// TIA Portal project "MIxProject" (V21)

(* hardware
DEVICE "S7-1500/ET200MP station_1"  S7-1500 station
   slot 0: "Rail_0"  Rack  6ES7 590-1***0-0AA0
   slot 1: "PLC_1"  CPU 1511-1 PN  6ES7 511-1AK02-0AB0  V2.9
      slot 3: "CPU display_1"  6ES7591-1AA00-0AA0
      slot 32768: "PROFINET interface_1"  X1
         slot 32769: "Port_1"  X1 P1
         slot 32770: "Port_2"  X1 P2
      slot 34817: "Virtual CP interface port_1"  Virtual CP interface port  Virtual CP interface port
DEVICE "HMI_1"  KTP700 Basic PN
   slot 0: "HMI_1"  KTP700 Basic PN  6AV2 123-2GB03-0AX0  17.0.0.0
   slot 1: "HMI_RT_1"  KTP700 Basic PN  6AV2 123-2GB03-0AX0  17.0.0.0
   slot 5: "HMI_1.IE_CP_1"  PROFINET Interface  17.0.0.0
      slot 1: "PROFINET Interface_1"  PROFINET Interface
         slot 1: "Port_1"  Port
*)

// ===== PLC "PLC_1"  CPU 1511-1 PN =====

VAR_GLOBAL   // PLC tag table "Default tag table"
   "valveA" AT %Q0.0 : Bool;
   "valveB" AT %Q0.1 : Bool;
   "valveC" AT %Q0.2 : Bool;
   "MIX" AT %Q0.3 : Bool;
   "TempSensor" AT %MD100 : Real;
   "LevelSensor" AT %MD200 : Real;
   "Start" AT %I0.4 : Bool;
   "Stop" AT %I0.5 : Bool;
   "Emergency" AT %I0.6 : Bool;
   "HeaterON/OFF" AT %M0.0 : Bool;
   "HeaterOutput" AT %MD300 : Real;
   "Setpoint" AT %MD4 : Real;
   "CurrentStep" AT %MW400 : Int;
END_VAR

DATA_BLOCK "FB_MixingSequence_DB"   // DB1
{ S7_Optimized_Access := 'TRUE' }
VERSION : 0.1
// stored: InstanceOfName FB_MixingSequence
"FB_MixingSequence"
BEGIN
END_DATA_BLOCK

DATA_BLOCK "sim_DB"   // DB3
{ S7_Optimized_Access := 'TRUE' }
VERSION : 0.1
// stored: InstanceOfName sim
"sim"
BEGIN
END_DATA_BLOCK

FUNCTION_BLOCK "FB_MixingSequence"   // FB1, GRAPH_PLUS
{ S7_Optimized_Access := 'TRUE' }
VERSION : 0.1
   VAR_INPUT
      OFF_SQ : Bool := false;   // Turn sequence off
      INIT_SQ : Bool := false;   // Set sequence to initial state
      ACK_EF : Bool := false;   // Acknowledge all errors and faults
      S_PREV : Bool := false;   // Output previous step in parameter S_NO
      S_NEXT : Bool := false;   // Indicate next step in parameter S_NO
      SW_AUTO : Bool := false;   // Automatic mode
      SW_TAP : Bool := false;   // Semiautomatic/switch with transition
      SW_TOP : Bool := false;   // Semiautomatic/ignore transition
      SW_MAN : Bool := false;   // Manual mode
      S_SEL : Int := 0;   // Select step to be output to S_NO
      S_ON : Bool := false;   // Activate step indicated in S_NO
      S_OFF : Bool := false;   // Disable step indicated in S_NO
      T_PUSH : Bool := false;   // Enable transition to switch in semi automatic mode
   END_VAR
   VAR_OUTPUT
      S_NO : Int := 0;   // Step number
      S_MORE : Bool := false;   // More steps are available and can be shown in S_NO
      S_ACTIVE : Bool := false;   // Step indicated in S_NO is active
      ERR_FLT : Bool := false;   // Interlock or supervision group error
      AUTO_ON : Bool := false;   // Automatic mode is active
      TAP_ON : Bool := false;   // Semiautomatic mode/step with transition enabled
      TOP_ON : Bool := false;   // Semiautomatic mode/ignore transition enabled
      MAN_ON : Bool := false;   // Manual mode is active
   END_VAR
   VAR
      HMI_INFO : Array[0..8] of UInt;
      IF_PAR : G7_IfParPlus_V6;
      RT_DATA : G7_RTDataPlus_V6;   // Internal data area
      Trans1 : G7_TransitionPlus_V6;   // Transition structure
      Trans2 : G7_TransitionPlus_V6;   // Transition structure
      Trans3 : G7_TransitionPlus_V6;   // Transition structure
      Trans4 : G7_TransitionPlus_V6;   // Transition structure
      Trans5 : G7_TransitionPlus_V6;   // Transition structure
      Step1 : G7_StepPlus_V6;   // Step structure
      Step2 : G7_StepPlus_V6;   // Step structure
      Step3 : G7_StepPlus_V6;   // Step structure
      Step4 : G7_StepPlus_V6;   // Step structure
      Step5 : G7_StepPlus_V6;   // Step structure
      SINI : Array[0..1] of USInt;
      LSTT : Array[0..4] of USInt;
      ATAJ : Array[0..4] of USInt;
      ATAB : Array[0..4] of USInt;
      PSTT : Array[0..4] of USInt;
      NSTT : Array[0..4] of USInt;
      ASSJ : Array[0..4] of USInt;
      ASSB : Array[0..4] of USInt;
      PTTS : Array[0..4] of USInt;
      NTTS : Array[0..4] of USInt;
      SW_SQTS : Array[0..4] of USInt;
      SWITCH : Array[0..0] of USInt;
      TVX : Array[0..1] of USInt;
      TTX : Array[0..1] of USInt;
      TSX : Array[0..1] of USInt;
      S00X : Array[0..1] of USInt;
      SOFFX : Array[0..1] of USInt;
      SONX : Array[0..1] of USInt;
      SAX : Array[0..1] of USInt;
      SERRX : Array[0..5] of USInt;
      SMX : Array[0..5] of USInt;
      S0X : Array[0..5] of USInt;
      S1X : Array[0..5] of USInt;
      IL_ALARM_INST : Diag_Alarm;
      SUP_ALARM_INST : Diag_Alarm;
      STEP_TIME_ALARM_INST : Diag_Alarm;
      IEC_TIMER_INST : IEC_TIMER;
      TRANSACTION_FLAG : Bool := false;
   END_VAR
   // SINI[0] := 2;
   // LSTT[0] := 255;
   // LSTT[1] := 255;
   // LSTT[2] := 255;
   // LSTT[3] := 255;
   // ATAJ[1] := 1;
   // ATAJ[2] := 2;
   // ATAJ[3] := 3;
   // ATAJ[4] := 4;
   // ATAB[1] := 1;
   // ATAB[2] := 2;
   // ATAB[3] := 3;
   // ATAB[4] := 4;
   // PSTT[1] := 1;
   // PSTT[2] := 2;
   // PSTT[3] := 3;
   // PSTT[4] := 4;
   // NSTT[0] := 1;
   // NSTT[1] := 2;
   // NSTT[2] := 3;
   // NSTT[3] := 4;
   // ASSJ[1] := 1;
   // ASSJ[2] := 2;
   // ASSJ[3] := 3;
   // ASSJ[4] := 4;
   // ASSB[1] := 1;
   // ASSB[2] := 2;
   // ASSB[3] := 3;
   // ASSB[4] := 4;
   // PTTS[0] := 255;
   // PTTS[2] := 1;
   // PTTS[3] := 2;
   // PTTS[4] := 3;
   // NTTS[1] := 1;
   // NTTS[2] := 2;
   // NTTS[3] := 3;
   // NTTS[4] := 4;
   // TVX[0] := 16#1;
   // TTX[0] := 16#1;
   // TSX[0] := 16#1;
   // S00X[0] := 16#1;
   // SOFFX[0] := 16#1;
   // SONX[0] := 16#1;
   // SAX[0] := 16#1;
   // SERRX[0] := 16#1;
   // SMX[0] := 16#1;
   // S0X[0] := 16#1;
   // S1X[0] := 16#1;
BEGIN
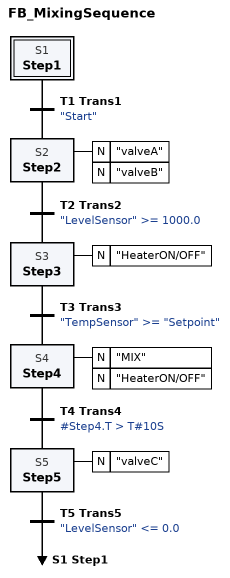
   // sequencer 1
   INITIAL_STEP Step1:   // S1, max time T#10S, warning time T#7S
   END_STEP
   TRANSITION Trans1 FROM Step1 TO Step2   // T1
      := "Start";
   END_TRANSITION
   STEP Step2:   // S2, max time T#10S, warning time T#7S
              N    "valveA"
              N    "valveB"
   END_STEP
   TRANSITION Trans2 FROM Step2 TO Step3   // T2
      := "LevelSensor" >= 1000.0;
   END_TRANSITION
   STEP Step3:   // S3, max time T#10S, warning time T#7S
              N    "HeaterON/OFF"
   END_STEP
   TRANSITION Trans3 FROM Step3 TO Step4   // T3
      := "TempSensor" >= "Setpoint";
   END_TRANSITION
   STEP Step4:   // S4, max time T#10S, warning time T#7S
              N    "MIX"
              N    "HeaterON/OFF"
   END_STEP
   TRANSITION Trans4 FROM Step4 TO Step5   // T4
      := #Step4.T > T#10S;
   END_TRANSITION
   STEP Step5:   // S5, max time T#10S, warning time T#7S
              N    "valveC"
   END_STEP
   TRANSITION Trans5 FROM Step5 TO Step1   // T5, jump
      := "LevelSensor" <= 0.0;
   END_TRANSITION
END_FUNCTION_BLOCK

FUNCTION_BLOCK "sim"   // FB2, SCL
{ S7_Optimized_Access := 'TRUE' }
VERSION : 0.1
BEGIN

   IF "valveA" OR "valveB" THEN
       "LevelSensor" := "LevelSensor" + 0.5;
   END_IF;

   IF "valveC" THEN
       "LevelSensor" := "LevelSensor" - 1.0;
   END_IF;


   IF "LevelSensor" > 1000.0 THEN
       "LevelSensor" := 1000.0;
   END_IF;
   IF "LevelSensor" < 0.0 THEN
       "LevelSensor" := 0.0;
   END_IF;


   IF "HeaterON/OFF" THEN
       "TempSensor" := "TempSensor" + ("HeaterOutput" * 0.01);
   ELSE
       "TempSensor" := "TempSensor" - 0.1; 
   END_IF;


   IF "TempSensor" > 120.0 THEN
       "TempSensor" := 120.0;
   END_IF;
   IF "TempSensor" < 0.0 THEN
       "TempSensor" := 0.0;
   END_IF;
END_FUNCTION_BLOCK

FUNCTION "fastreset" : Void   // FC1, SCL
{ S7_Optimized_Access := 'TRUE' }
VERSION : 0.1
BEGIN
   "valveA" := FALSE;
   "valveB" := FALSE;
   "MIX" := FALSE;
   "HeaterON/OFF" := FALSE;
   IF "LevelSensor" > 0 THEN
       "valveC" := TRUE;
   ELSE
       "valveC" := FALSE;
   END_IF;
END_FUNCTION

ORGANIZATION_BLOCK "Main"   // OB1, LAD, ProgramCycle
TITLE = "Main Program Sweep (Cycle)"
{ S7_Optimized_Access := 'TRUE' }
VERSION : 0.1
   VAR_INPUT
      Initial_Call : Bool;   // Initial call of this OB
      Remanence : Bool;   // =True, if remanent data are available
   END_VAR
BEGIN

REGION Network 1
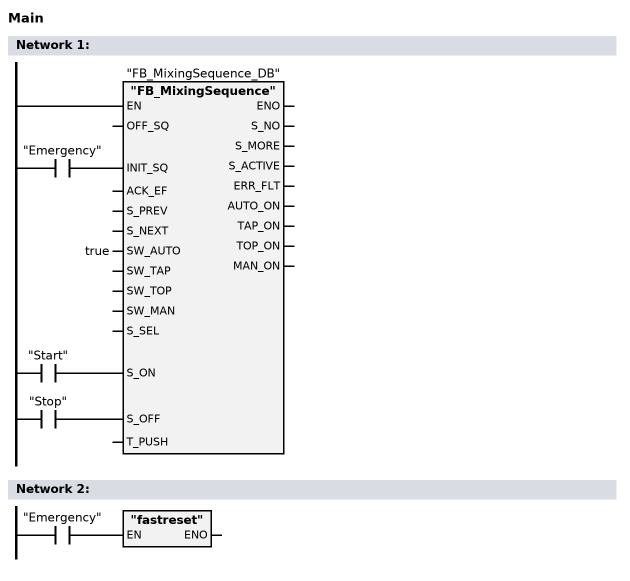
   RUNG wire#powerrail
      "FB_MixingSequence_DB"(INIT_SQ := wire#w1, S_ON := wire#w2, S_OFF := wire#w3, OFF_SQ :=, ACK_EF :=, S_PREV :=, S_NEXT :=, SW_AUTO := true, SW_TAP :=, SW_TOP :=, SW_MAN :=, S_SEL :=, T_PUSH :=, S_NO =>, S_MORE =>, S_ACTIVE =>, ERR_FLT =>, AUTO_ON =>, TAP_ON =>, TOP_ON =>, MAN_ON =>)
   END_RUNG
   RUNG wire#powerrail
      Contact( "Emergency" )
   END_RUNG wire#w1
   RUNG wire#powerrail
      Contact( "Start" )
   END_RUNG wire#w2
   RUNG wire#powerrail
      Contact( "Stop" )
   END_RUNG wire#w3
   // the same network as SCL:
   "FB_MixingSequence_DB"(INIT_SQ := "Emergency", SW_AUTO := true, S_ON := "Start", S_OFF := "Stop");   // "FB_MixingSequence"
END_REGION

REGION Network 2
   RUNG wire#powerrail
      Contact( "Emergency" )
      "fastreset"()
   END_RUNG
   // the same network as SCL:
   IF "Emergency" THEN "fastreset"(); END_IF;
END_REGION

REGION Network 3 (SCL)
   IF "Emergency" OR "Stop" THEN
       "CurrentStep" := 0;
   ELSE
       "CurrentStep" := UINT_TO_INT("FB_MixingSequence_DB".S_NO);
   END_IF;
END_REGION
END_ORGANIZATION_BLOCK

ORGANIZATION_BLOCK "CyclicInterrupt"   // OB30, FBD, CyclicInterrupt
{ S7_Optimized_Access := 'TRUE' }
VERSION : 0.1
   VAR_INPUT
      Initial_Call : Bool;   // Initial call of this OB
      Event_Count : Int;   // Events discarded
   END_VAR
BEGIN

REGION Network 1
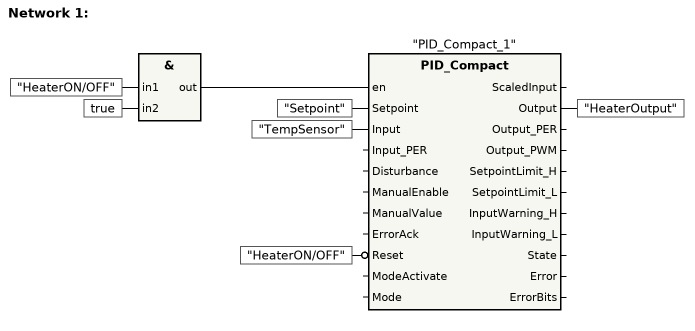
   IF "HeaterON/OFF" AND true THEN
       "PID_Compact_1"(Setpoint := "Setpoint",   // PID_Compact
                       Input := "TempSensor",
                       Reset := NOT "HeaterON/OFF",
                       Output => "HeaterOutput");
   END_IF;
END_REGION

REGION Network 2 (SCL)
   IF "valveA" OR "valveB" THEN
       "LevelSensor" := "LevelSensor" + 10.0;
   END_IF;
   IF "valveC" THEN
       "LevelSensor" := "LevelSensor" - 10.0;
   END_IF;


   IF "LevelSensor" > 1000.0 THEN
       "LevelSensor" := 1000.0;
   END_IF;
   IF "LevelSensor" < 0.0 THEN
       "LevelSensor" := 0.0;
   END_IF;


   IF "HeaterON/OFF" THEN
       "TempSensor" := "TempSensor" +
       ("HeaterOutput" * 0.001 * (120.0 - "TempSensor") / 120.0);
   ELSE
       "TempSensor" := "TempSensor" - 0.05;
       "HeaterOutput" := 0;
   END_IF;


   IF "TempSensor" > 120.0 THEN
       "TempSensor" := 120.0;
   END_IF;
   IF "TempSensor" < 0.0 THEN
       "TempSensor" := 0.0;
   END_IF;
END_REGION
END_ORGANIZATION_BLOCK

(* ===== HMI "HMI_RT_1" =====
system functions are stored by id; their names below are inferred from use
connection "HMI_Connection_1": ETHERNET, SMART_S7_1500_OMS

HMI tags "Default tag table"
   "Tag_ScreenNumber" : UInt, internal
   "Start" : Bool = PLC Start AT %I0.4, 1 s
   "Stop" : Bool = PLC Stop AT %I0.5, 1 s
   "Emergency" : Bool = PLC Emergency AT %I0.6, 1 s
   "LevelSensor" : Real = PLC LevelSensor AT %MD200, 1 s
   "TempSensor" : Real = PLC TempSensor AT %MD100, 1 s
   "Setpoint" : Real = PLC Setpoint AT %MD4, 1 s
   "CurrentStep" : Int = PLC CurrentStep AT %MW400, 1 s
   "HeaterOutput" : Real = PLC HeaterOutput AT %MD300, 1 s

text list "StepNames": 1 'Waiting'; 2 'Filling'; 3 'Heating'; 4 'Mixing'; 5 'Drain'; 0 'Emergency/Stop'

Template "Template_1" 800x480
   Button "Exit" at 714,429 size 71x50; TextOff 'Exit'; PictureOff "ExitRuntime_KTP700_Basic_PN_TR"; PictureOn "ExitRuntime_KTP700_Basic_PN_TR"
      on Release: StopRuntime(0)
   Button "Template_Button" at 614,429 size 71x50; TextOff 'Text'
   Button "Template_Button_1" at 514,429 size 71x50; TextOff 'Text'
   Button "Template_Button_2" at 414,429 size 71x50; TextOff 'Text'
   Button "Template_Button_3" at 314,429 size 71x50; TextOff 'Text'
   Button "Template_Button_4" at 214,429 size 71x50; TextOff 'Text'
   Button "Alarms" at 114,429 size 71x50; TextOff 'Alarms'; PictureOff "AlarmDisplay_KTP700_Basic_PN_TR"; PictureOn "AlarmDisplay_KTP700_Basic_PN_TR"
      on Release: function_ef3f5d25("Alarm window_Unacknowledged", -1)
   Button "Start screen" at 14,429 size 71x50; TextOff 'Start screen'; PictureOff "NavigateHome_KTP700_Basic_PN_TR"; PictureOn "NavigateHome_KTP700_Basic_PN_TR"
      on Release: ActivateScreen("Root screen", 0)
   SymbolicIOField "Symbolic_IO_Field_Screen" at 93,9 size 600x33; TextOff '0'; TextOn '1'; TextList "StepNames"
      ProcessValue <- "Tag_ScreenNumber"
      on Change: ActivateScreenByNumber("Tag_ScreenNumber", 0)
   DateTimeField "HmiScreenItemData" at 695,25 size 105x25
   DateTimeField "HmiScreenItemData_1" at 695,0 size 105x25
   GraphicView "Logo" at 0,0 size 91x51; Picture "Logo of HMI_1"

screen "Root screen" 800x480, template "Template_1"
   on GenerateScreen: SetTag("Tag_ScreenNumber", 1)
   TextField "HmiScreenItemData" at 80,225 size 640x25; Text 'Welcome to HMI_1 (KTP700 Basic+ PN)!'
   Button "Button_1" at 328,278 size 130x32; TextOff 'main screen'
      on Click: ActivateScreen("Screen_1", 0)

screen "Screen_1" 800x480
   Button "Button_1" at 18,427 size 96x32; TextOff 'Start'
      on Press: SetBit("Start")
      on Release: ResetBit("Start")
   Button "Button_2" at 135,427 size 96x32; TextOff 'Stop'
      on Press: SetBit("Stop")
      on Release: ResetBit("Stop")
   Button "Button_3" at 250,427 size 96x32; TextOff 'Emergency'
      on Press: SetBit("Emergency")
      on Release: ResetBit("Emergency")
   Bar "Bar_1" at 20,71 size 249x328; MinimumValue 0; MaximumValue 1000
      ProcessValue <- "LevelSensor"
   IOField "I/O field_1" at 307,34 size 111x41; FormatPattern 99.9
      ProcessValue <- "TempSensor"
   IOField "I/O field_3" at 437,33 size 114x42; FormatPattern 99.9
      ProcessValue <- "Setpoint"
   TextField "Text field_1" at 301,12 size 112x23; Text 'Temperature'
   TextField "Text field_3" at 435,11 size 74x23; Text 'Setpoint'
   SymbolicIOField "Symbolic I/O field_1" at 17,18 size 255x32; TextOff '0'; TextOn '1'; TextList "StepNames"
      ProcessValue <- "CurrentStep"
   TrendView "Trend view_1" at 307,84 size 439x314
   IOField "I/O field_2" at 564,32 size 114x42; FormatPattern 99.9
      ProcessValue <- "HeaterOutput"
   TextField "Text field_2" at 562,10 size 117x23; Text 'HeaterOutput'
*)